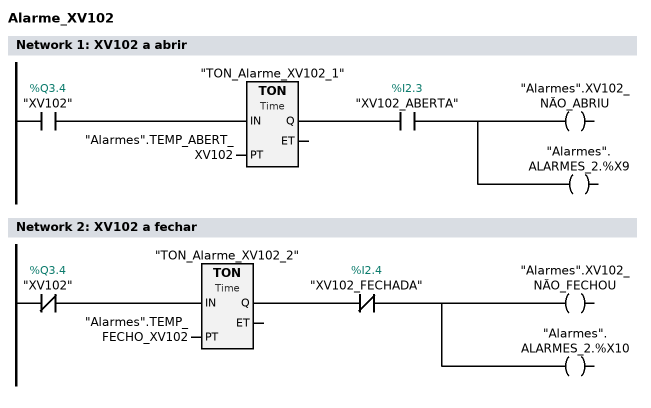
   RUNG wire#powerrail
      Contact( "XV102" )
      { S7_Templates := "time_type := Time" } "TON_Alarme_XV102_1".TON(pt := "Alarmes".TEMP_ABERT_XV102, et =>)
      Contact( "XV102_ABERTA" )
      wire#w1
      Coil( "Alarmes".XV102_NÃO_ABRIU )
   END_RUNG
   RUNG wire#w1
      Coil( "Alarmes".ALARMES_2.%X9 )
   END_RUNG
   // the same network as SCL:
   "TON_Alarme_XV102_1".TON(IN := "XV102", PT := "Alarmes".TEMP_ABERT_XV102);
   "Alarmes".XV102_NÃO_ABRIU := "TON_Alarme_XV102_1".Q AND "XV102_ABERTA";
   "Alarmes".ALARMES_2.%X9 := "Alarmes".XV102_NÃO_ABRIU;
END_REGION

REGION Network 2: XV102 a fechar
   RUNG wire#powerrail
      I_Contact( "XV102" )
      { S7_Templates := "time_type := Time" } "TON_Alarme_XV102_2".TON(pt := "Alarmes".TEMP_FECHO_XV102, et =>)
      I_Contact( "XV102_FECHADA" )
      wire#w1
      Coil( "Alarmes".XV102_NÃO_FECHOU )
   END_RUNG
   RUNG wire#w1
      Coil( "Alarmes".ALARMES_2.%X10 )
   END_RUNG
   // the same network as SCL:
   "TON_Alarme_XV102_2".TON(IN := NOT "XV102", PT := "Alarmes".TEMP_FECHO_XV102);
   "Alarmes".XV102_NÃO_FECHOU := "TON_Alarme_XV102_2".Q AND NOT "XV102_FECHADA";
   "Alarmes".ALARMES_2.%X10 := "Alarmes".XV102_NÃO_FECHOU;
END_REGION
END_FUNCTION

FUNCTION "Reinício_Ciclo" : Void   // FC19, LAD
{ S7_Optimized_Access := 'TRUE' }
VERSION : 0.1
// stored: AutoNumber true, IsIECCheckEnabled false, SetENOAutomatically false, UDAEnableTagReadback false
   VAR_TEMP   // added for the SCL form of the ladder/FBD networks
      _w1 : Bool;
   END_VAR
BEGIN

REGION Network 1: Ativa etapa 1 e faz reset às restantes do ciclo de tratamento
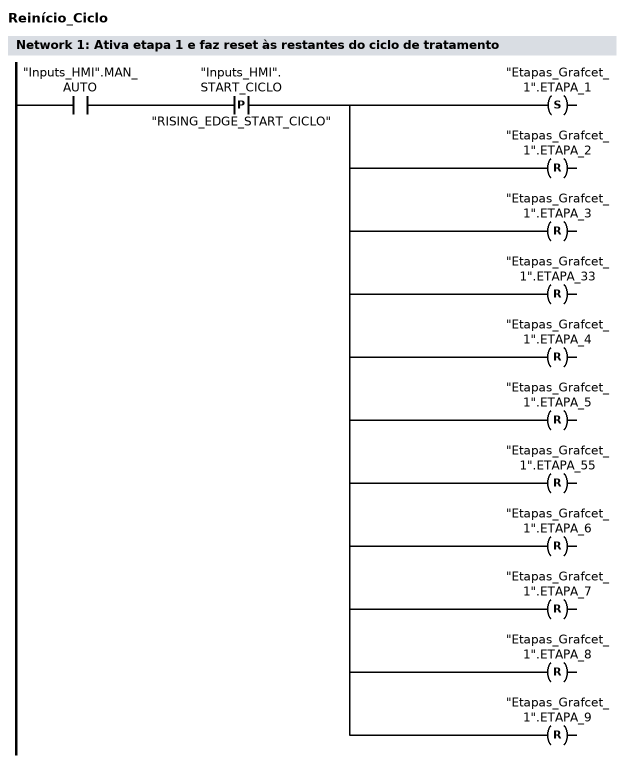
   RUNG wire#powerrail
      Contact( "Inputs_HMI".MAN_AUTO )
      P_Contact(operand := "Inputs_HMI".START_CICLO, bit := "RISING_EDGE_START_CICLO")
      wire#w1
      S_Coil( "Etapas_Grafcet_1".ETAPA_1 )
   END_RUNG
   RUNG wire#w1
      R_Coil( "Etapas_Grafcet_1".ETAPA_2 )
   END_RUNG
   RUNG wire#w1
      R_Coil( "Etapas_Grafcet_1".ETAPA_3 )
   END_RUNG
   RUNG wire#w1
      R_Coil( "Etapas_Grafcet_1".ETAPA_33 )
   END_RUNG
   RUNG wire#w1
      R_Coil( "Etapas_Grafcet_1".ETAPA_4 )
   END_RUNG
   RUNG wire#w1
      R_Coil( "Etapas_Grafcet_1".ETAPA_5 )
   END_RUNG
   RUNG wire#w1
      R_Coil( "Etapas_Grafcet_1".ETAPA_55 )
   END_RUNG
   RUNG wire#w1
      R_Coil( "Etapas_Grafcet_1".ETAPA_6 )
   END_RUNG
   RUNG wire#w1
      R_Coil( "Etapas_Grafcet_1".ETAPA_7 )
   END_RUNG
   RUNG wire#w1
      R_Coil( "Etapas_Grafcet_1".ETAPA_8 )
   END_RUNG
   RUNG wire#w1
      R_Coil( "Etapas_Grafcet_1".ETAPA_9 )
   END_RUNG
   // the same network as SCL:
   #_w1 := "Inputs_HMI".MAN_AUTO AND "Inputs_HMI".START_CICLO AND NOT "RISING_EDGE_START_CICLO";   // rising edge of "Inputs_HMI".START_CICLO
   "RISING_EDGE_START_CICLO" := "Inputs_HMI".START_CICLO;
   IF #_w1 THEN
       "Etapas_Grafcet_1".ETAPA_1 := TRUE;
       "Etapas_Grafcet_1".ETAPA_2 := FALSE;
       "Etapas_Grafcet_1".ETAPA_3 := FALSE;
       "Etapas_Grafcet_1".ETAPA_33 := FALSE;
       "Etapas_Grafcet_1".ETAPA_4 := FALSE;
       "Etapas_Grafcet_1".ETAPA_5 := FALSE;
       "Etapas_Grafcet_1".ETAPA_55 := FALSE;
       "Etapas_Grafcet_1".ETAPA_6 := FALSE;
       "Etapas_Grafcet_1".ETAPA_7 := FALSE;
       "Etapas_Grafcet_1".ETAPA_8 := FALSE;
       "Etapas_Grafcet_1".ETAPA_9 := FALSE;
   END_IF;
END_REGION
END_FUNCTION

FUNCTION "Estab_Níveis" : Void   // FC20, LAD
TITLE = Protege equipamentos e evita transbordo em modo manual
{ S7_Optimized_Access := 'TRUE' }
VERSION : 0.1
// stored: AutoNumber true, IsIECCheckEnabled false, SetENOAutomatically false, UDAEnableTagReadback false
BEGIN

REGION Network 1: LSL001
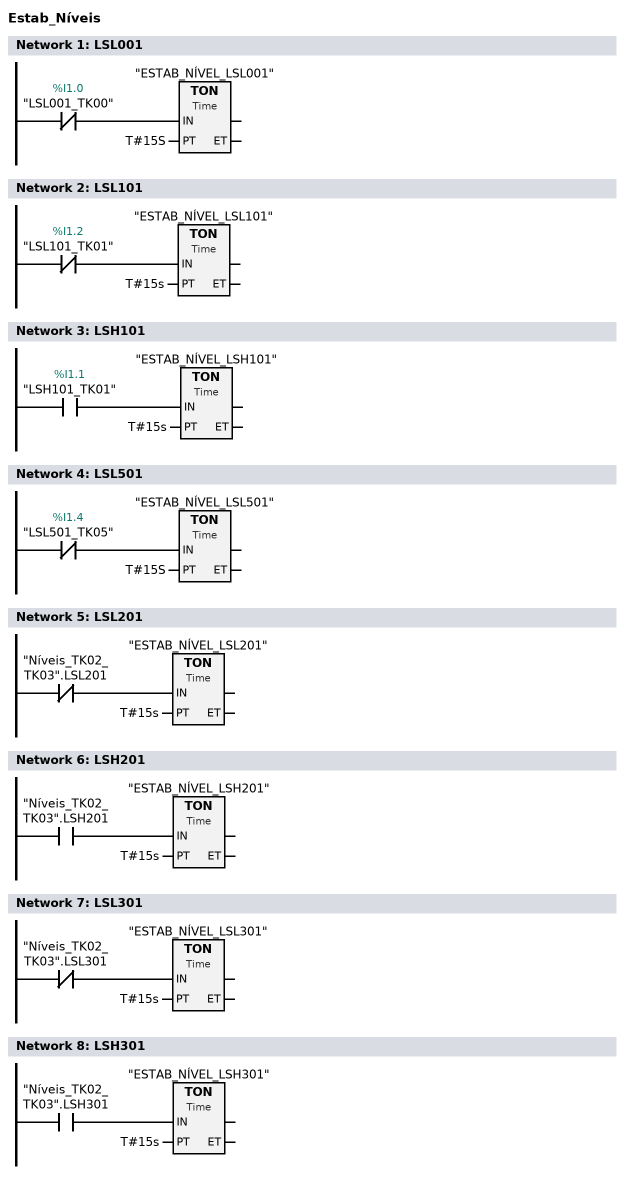
   RUNG wire#powerrail
      I_Contact( "LSL001_TK00" )
      { S7_Templates := "time_type := Time" } "ESTAB_NÍVEL_LSL001".TON(pt := T#15S, et =>)
   END_RUNG
   // the same network as SCL:
   "ESTAB_NÍVEL_LSL001".TON(IN := NOT "LSL001_TK00", PT := T#15S);
END_REGION

REGION Network 2: LSL101
   RUNG wire#powerrail
      I_Contact( "LSL101_TK01" )
      { S7_Templates := "time_type := Time" } "ESTAB_NÍVEL_LSL101".TON(pt := T#15s, et =>)
   END_RUNG
   // the same network as SCL:
   "ESTAB_NÍVEL_LSL101".TON(IN := NOT "LSL101_TK01", PT := T#15s);
END_REGION

REGION Network 3: LSH101
   RUNG wire#powerrail
      Contact( "LSH101_TK01" )
      { S7_Templates := "time_type := Time" } "ESTAB_NÍVEL_LSH101".TON(pt := T#15s, et =>)
   END_RUNG
   // the same network as SCL:
   "ESTAB_NÍVEL_LSH101".TON(IN := "LSH101_TK01", PT := T#15s);
END_REGION

REGION Network 4: LSL501
   RUNG wire#powerrail
      I_Contact( "LSL501_TK05" )
      { S7_Templates := "time_type := Time" } "ESTAB_NÍVEL_LSL501".TON(pt := T#15S, et =>)
   END_RUNG
   // the same network as SCL:
   "ESTAB_NÍVEL_LSL501".TON(IN := NOT "LSL501_TK05", PT := T#15S);
END_REGION

REGION Network 5: LSL201
   RUNG wire#powerrail
      I_Contact( "Níveis_TK02_TK03".LSL201 )
      { S7_Templates := "time_type := Time" } "ESTAB_NÍVEL_LSL201".TON(pt := T#15s, et =>)
   END_RUNG
   // the same network as SCL:
   "ESTAB_NÍVEL_LSL201".TON(IN := NOT "Níveis_TK02_TK03".LSL201, PT := T#15s);
END_REGION

REGION Network 6: LSH201
   RUNG wire#powerrail
      Contact( "Níveis_TK02_TK03".LSH201 )
      { S7_Templates := "time_type := Time" } "ESTAB_NÍVEL_LSH201".TON(pt := T#15s, et =>)
   END_RUNG
   // the same network as SCL:
   "ESTAB_NÍVEL_LSH201".TON(IN := "Níveis_TK02_TK03".LSH201, PT := T#15s);
END_REGION

REGION Network 7: LSL301
   RUNG wire#powerrail
      I_Contact( "Níveis_TK02_TK03".LSL301 )
      { S7_Templates := "time_type := Time" } "ESTAB_NÍVEL_LSL301".TON(pt := T#15s, et =>)
   END_RUNG
   // the same network as SCL:
   "ESTAB_NÍVEL_LSL301".TON(IN := NOT "Níveis_TK02_TK03".LSL301, PT := T#15s);
END_REGION

REGION Network 8: LSH301
   RUNG wire#powerrail
      Contact( "Níveis_TK02_TK03".LSH301 )
      { S7_Templates := "time_type := Time" } "ESTAB_NÍVEL_LSH301".TON(pt := T#15s, et =>)
   END_RUNG
   // the same network as SCL:
   "ESTAB_NÍVEL_LSH301".TON(IN := "Níveis_TK02_TK03".LSH301, PT := T#15s);
END_REGION
END_FUNCTION

FUNCTION "Contador_de_Ciclos" : Void   // FC21, LAD
{ S7_Optimized_Access := 'TRUE' }
VERSION : 0.1
// stored: AutoNumber true, IsIECCheckEnabled false, SetENOAutomatically false, UDAEnableTagReadback false
BEGIN

REGION Network 1: Conta o número de ciclos de tratamento
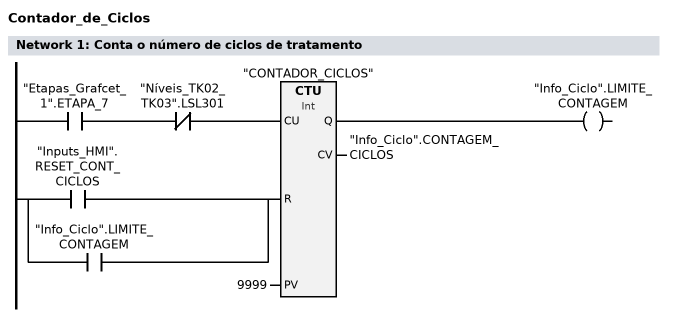
   RUNG wire#powerrail
      Contact( "Etapas_Grafcet_1".ETAPA_7 )
      I_Contact( "Níveis_TK02_TK03".LSL301 )
      { S7_Templates := "value_type := Int" } "CONTADOR_CICLOS".CTU(r := wire#w1, pv := 9999, cv => "Info_Ciclo".CONTAGEM_CICLOS)
      Coil( "Info_Ciclo".LIMITE_CONTAGEM )
   END_RUNG
   RUNG wire#powerrail
      Contact( "Inputs_HMI".RESET_CONT_CICLOS )
   END_RUNG wire#w1
   RUNG wire#powerrail
      Contact( "Info_Ciclo".LIMITE_CONTAGEM )
   END_RUNG wire#w1
   // the same network as SCL:
   "CONTADOR_CICLOS".CTU(CU := "Etapas_Grafcet_1".ETAPA_7 AND NOT "Níveis_TK02_TK03".LSL301,
                         R := "Inputs_HMI".RESET_CONT_CICLOS OR "Info_Ciclo".LIMITE_CONTAGEM,
                         PV := 9999,
                         CV => "Info_Ciclo".CONTAGEM_CICLOS);
   "Info_Ciclo".LIMITE_CONTAGEM := "CONTADOR_CICLOS".Q;
END_REGION
END_FUNCTION

FUNCTION "Reset_Etapas_Iniciais" : Void   // FC23, LAD
TITLE = Reset às etapas inicias em caso de falha de energia, de modo e continuar o processo do ponto onde estava
{ S7_Optimized_Access := 'TRUE' }
VERSION : 0.1
// stored: AutoNumber true, IsIECCheckEnabled false, SetENOAutomatically false, UDAEnableTagReadback false
BEGIN

REGION Network 1: Reset etapa 1
   // as etapas 3, 33 e 7 não precisam nem devem fazer reset à etapa 1. Já é feito indiretamente no FC4
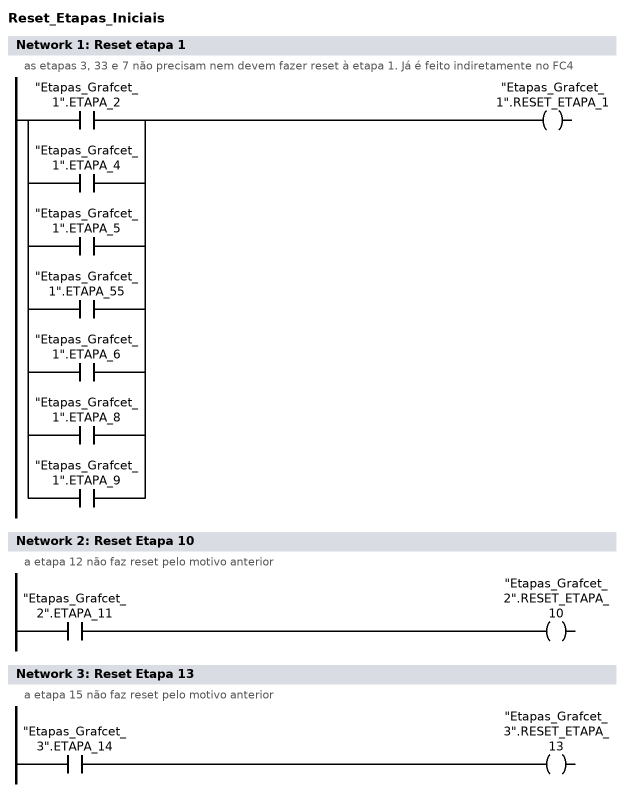
   RUNG wire#powerrail
      Contact( "Etapas_Grafcet_1".ETAPA_2 )
      wire#w1
      Coil( "Etapas_Grafcet_1".RESET_ETAPA_1 )
   END_RUNG
   RUNG wire#powerrail
      Contact( "Etapas_Grafcet_1".ETAPA_4 )
   END_RUNG wire#w1
   RUNG wire#powerrail
      Contact( "Etapas_Grafcet_1".ETAPA_5 )
   END_RUNG wire#w1
   RUNG wire#powerrail
      Contact( "Etapas_Grafcet_1".ETAPA_55 )
   END_RUNG wire#w1
   RUNG wire#powerrail
      Contact( "Etapas_Grafcet_1".ETAPA_6 )
   END_RUNG wire#w1
   RUNG wire#powerrail
      Contact( "Etapas_Grafcet_1".ETAPA_8 )
   END_RUNG wire#w1
   RUNG wire#powerrail
      Contact( "Etapas_Grafcet_1".ETAPA_9 )
   END_RUNG wire#w1
   // the same network as SCL:
   "Etapas_Grafcet_1".RESET_ETAPA_1 := "Etapas_Grafcet_1".ETAPA_2 OR "Etapas_Grafcet_1".ETAPA_4 OR "Etapas_Grafcet_1".ETAPA_5 OR "Etapas_Grafcet_1".ETAPA_55 OR "Etapas_Grafcet_1".ETAPA_6 OR "Etapas_Grafcet_1".ETAPA_8 OR "Etapas_Grafcet_1".ETAPA_9;
END_REGION

REGION Network 2: Reset Etapa 10
   // a etapa 12 não faz reset pelo motivo anterior
   RUNG wire#powerrail
      Contact( "Etapas_Grafcet_2".ETAPA_11 )
      Coil( "Etapas_Grafcet_2".RESET_ETAPA_10 )
   END_RUNG
   // the same network as SCL:
   "Etapas_Grafcet_2".RESET_ETAPA_10 := "Etapas_Grafcet_2".ETAPA_11;
END_REGION

REGION Network 3: Reset Etapa 13
   // a etapa 15 não faz reset pelo motivo anterior
   RUNG wire#powerrail
      Contact( "Etapas_Grafcet_3".ETAPA_14 )
      Coil( "Etapas_Grafcet_3".RESET_ETAPA_13 )
   END_RUNG
   // the same network as SCL:
   "Etapas_Grafcet_3".RESET_ETAPA_13 := "Etapas_Grafcet_3".ETAPA_14;
END_REGION
END_FUNCTION

DATA_BLOCK "CONTADOR_CICLOS"   // DB25
{ S7_Optimized_Access := 'TRUE' }
// stored: AutoNumber true, InstanceOfName IEC_COUNTER, OfSystemLibElement IEC_COUNTER, OfSystemLibVersion 1.0
"IEC_COUNTER"
   // VAR RETAIN
   //    CU : Bool;
   //    CD : Bool;
   //    R : Bool;
   //    LD : Bool;
   //    QU : Bool;
   //    QD : Bool;
   //    PV : Int;
   //    CV : Int;
   // END_VAR
BEGIN
END_DATA_BLOCK

DATA_BLOCK "ESTAB_NÍVEL_LSH101"   // DB17
{ S7_Optimized_Access := 'TRUE' }
// stored: AutoNumber true, InstanceOfName IEC_TIMER, OfSystemLibElement IEC_TIMER, OfSystemLibVersion 1.0
"IEC_TIMER"
   // VAR
   //    PT : Time;
   //    ET { ExternalWritable := 'False'} : Time;
   //    IN : Bool;
   //    Q { ExternalWritable := 'False'} : Bool;
   // END_VAR
BEGIN
END_DATA_BLOCK

DATA_BLOCK "ESTAB_NÍVEL_LSH201"   // DB21
{ S7_Optimized_Access := 'TRUE' }
// stored: AutoNumber true, InstanceOfName IEC_TIMER, OfSystemLibElement IEC_TIMER, OfSystemLibVersion 1.0
"IEC_TIMER"
   // VAR
   //    PT : Time;
   //    ET { ExternalWritable := 'False'} : Time;
   //    IN : Bool;
   //    Q { ExternalWritable := 'False'} : Bool;
   // END_VAR
BEGIN
END_DATA_BLOCK

DATA_BLOCK "ESTAB_NÍVEL_LSH301"   // DB23
{ S7_Optimized_Access := 'TRUE' }
// stored: AutoNumber true, InstanceOfName IEC_TIMER, OfSystemLibElement IEC_TIMER, OfSystemLibVersion 1.0
"IEC_TIMER"
   // VAR
   //    PT : Time;
   //    ET { ExternalWritable := 'False'} : Time;
   //    IN : Bool;
   //    Q { ExternalWritable := 'False'} : Bool;
   // END_VAR
BEGIN
END_DATA_BLOCK

DATA_BLOCK "ESTAB_NÍVEL_LSL001"   // DB19
{ S7_Optimized_Access := 'TRUE' }
// stored: AutoNumber true, InstanceOfName IEC_TIMER, OfSystemLibElement IEC_TIMER, OfSystemLibVersion 1.0
"IEC_TIMER"
   // VAR
   //    PT : Time;
   //    ET { ExternalWritable := 'False'} : Time;
   //    IN : Bool;
   //    Q { ExternalWritable := 'False'} : Bool;
   // END_VAR
BEGIN
END_DATA_BLOCK

DATA_BLOCK "ESTAB_NÍVEL_LSL101"   // DB20
{ S7_Optimized_Access := 'TRUE' }
// stored: AutoNumber true, InstanceOfName IEC_TIMER, OfSystemLibElement IEC_TIMER, OfSystemLibVersion 1.0
"IEC_TIMER"
   // VAR
   //    PT : Time;
   //    ET { ExternalWritable := 'False'} : Time;
   //    IN : Bool;
   //    Q { ExternalWritable := 'False'} : Bool;
   // END_VAR
BEGIN
END_DATA_BLOCK

DATA_BLOCK "ESTAB_NÍVEL_LSL201"   // DB22
{ S7_Optimized_Access := 'TRUE' }
// stored: AutoNumber true, InstanceOfName IEC_TIMER, OfSystemLibElement IEC_TIMER, OfSystemLibVersion 1.0
"IEC_TIMER"
   // VAR
   //    PT : Time;
   //    ET { ExternalWritable := 'False'} : Time;
   //    IN : Bool;
   //    Q { ExternalWritable := 'False'} : Bool;
   // END_VAR
BEGIN
END_DATA_BLOCK

DATA_BLOCK "ESTAB_NÍVEL_LSL301"   // DB24
{ S7_Optimized_Access := 'TRUE' }
// stored: AutoNumber true, InstanceOfName IEC_TIMER, OfSystemLibElement IEC_TIMER, OfSystemLibVersion 1.0
"IEC_TIMER"
   // VAR
   //    PT : Time;
   //    ET { ExternalWritable := 'False'} : Time;
   //    IN : Bool;
   //    Q { ExternalWritable := 'False'} : Bool;
   // END_VAR
BEGIN
END_DATA_BLOCK

DATA_BLOCK "ESTAB_NÍVEL_LSL501"   // DB18
{ S7_Optimized_Access := 'TRUE' }
// stored: AutoNumber true, InstanceOfName IEC_TIMER, OfSystemLibElement IEC_TIMER, OfSystemLibVersion 1.0
"IEC_TIMER"
   // VAR
   //    PT : Time;
   //    ET { ExternalWritable := 'False'} : Time;
   //    IN : Bool;
   //    Q { ExternalWritable := 'False'} : Bool;
   // END_VAR
BEGIN
END_DATA_BLOCK

DATA_BLOCK "TM0"   // DB5
{ S7_Optimized_Access := 'TRUE' }
// stored: AutoNumber true, InstanceOfName IEC_TIMER, OfSystemLibElement IEC_TIMER, OfSystemLibVersion 1.0
"IEC_TIMER"
   // VAR
   //    PT : Time;
   //    ET { ExternalWritable := 'False'} : Time;
   //    IN : Bool;
   //    Q { ExternalWritable := 'False'} : Bool;
   // END_VAR
BEGIN
END_DATA_BLOCK

DATA_BLOCK "TM1"   // DB6
{ S7_Optimized_Access := 'TRUE' }
// stored: AutoNumber true, InstanceOfName IEC_TIMER, OfSystemLibElement IEC_TIMER, OfSystemLibVersion 1.0
"IEC_TIMER"
   // VAR
   //    PT : Time;
   //    ET { ExternalWritable := 'False'} : Time;
   //    IN : Bool;
   //    Q { ExternalWritable := 'False'} : Bool;
   // END_VAR
BEGIN
END_DATA_BLOCK

DATA_BLOCK "TM2"   // DB7
{ S7_Optimized_Access := 'TRUE' }
// stored: AutoNumber true, InstanceOfName IEC_TIMER, OfSystemLibElement IEC_TIMER, OfSystemLibVersion 1.0
"IEC_TIMER"
   // VAR
   //    PT : Time;
   //    ET { ExternalWritable := 'False'} : Time;
   //    IN : Bool;
   //    Q { ExternalWritable := 'False'} : Bool;
   // END_VAR
BEGIN
END_DATA_BLOCK

DATA_BLOCK "TM3"   // DB8
{ S7_Optimized_Access := 'TRUE' }
// stored: AutoNumber true, InstanceOfName IEC_TIMER, OfSystemLibElement IEC_TIMER, OfSystemLibVersion 1.0
"IEC_TIMER"
   // VAR
   //    PT : Time;
   //    ET { ExternalWritable := 'False'} : Time;
   //    IN : Bool;
   //    Q { ExternalWritable := 'False'} : Bool;
   // END_VAR
BEGIN
END_DATA_BLOCK

DATA_BLOCK "TON_Alarme_XV102_1"   // DB16
{ S7_Optimized_Access := 'TRUE' }
// stored: AutoNumber true, InstanceOfName IEC_TIMER, OfSystemLibElement IEC_TIMER, OfSystemLibVersion 1.0
"IEC_TIMER"
   // VAR
   //    PT : Time;
   //    ET { ExternalWritable := 'False'} : Time;
   //    IN : Bool;
   //    Q { ExternalWritable := 'False'} : Bool;
   // END_VAR
BEGIN
END_DATA_BLOCK

DATA_BLOCK "TON_Alarme_XV102_2"   // DB26
{ S7_Optimized_Access := 'TRUE' }
// stored: AutoNumber true, InstanceOfName IEC_TIMER, OfSystemLibElement IEC_TIMER, OfSystemLibVersion 1.0
"IEC_TIMER"
   // VAR
   //    PT : Time;
   //    ET { ExternalWritable := 'False'} : Time;
   //    IN : Bool;
   //    Q { ExternalWritable := 'False'} : Bool;
   // END_VAR
BEGIN
END_DATA_BLOCK

DATA_BLOCK "T_DOS_COAGULANTE"   // DB9
{ S7_Optimized_Access := 'TRUE' }
// stored: AutoNumber true, InstanceOfName IEC_TIMER, OfSystemLibElement IEC_TIMER, OfSystemLibVersion 1.0
"IEC_TIMER"
   // VAR RETAIN
   //    PT : Time;
   //    ET { ExternalWritable := 'False'} : Time;
   //    IN : Bool;
   //    Q { ExternalWritable := 'False'} : Bool;
   // END_VAR
BEGIN
END_DATA_BLOCK

DATA_BLOCK "T_HISTERESE"   // DB2
{ S7_Optimized_Access := 'TRUE' }
// stored: AutoNumber true, InstanceOfName IEC_TIMER, OfSystemLibElement IEC_TIMER, OfSystemLibVersion 1.0
"IEC_TIMER"
   // VAR
   //    PT : Time;
   //    ET { ExternalWritable := 'False'} : Time;
   //    IN : Bool;
   //    Q { ExternalWritable := 'False'} : Bool;
   // END_VAR
BEGIN
END_DATA_BLOCK
